{attribute 'GeneratedUsingTerminal: EL3403-0000-0023'}
{attribute addProperty BoxType "EL3403-0000-0023"}
{attribute addProperty Id "IndexAT %Q*USINT1"}
{attribute addProperty CRC "3858488880"}
{attribute addProperty Size "1"}
TYPE PM_Outputs_Channel_E5FBDE30 :
STRUCT
	{attribute addProperty Name "Index"}
	Index AT %Q* : USINT;
END_STRUCT
END_TYPE

(* stored: Version 1.2.0.0, ProductVersion 3.1.4024.9
   DUT PM_Outputs_Channel_E5FBDE30: Id {388b80d2-1c76-0230-274b-81af7f87c624} *)
